(* Logix 5000 project; controller TORQUE Emulate 5570 rev 33.11; software revision 33.00 *)

TASK MainTask (continuous, watchdog 500 ms) : MainProgram, Emulation

MODULES
   Local : Emulate 5570 (ICP 2, rev 33.11)
       : 1756-IB16 (ICP 3, rev 3.1, Input RPI 20 ms)
       : vendor 1 type 7 code 16 (ICP 4, rev 3.1, Output RPI 20 ms)
       : 1756-IF8 (ICP 5, rev 1.1, Input RPI 100 ms)
END_MODULES

PROGRAM Emulation   (* main routine Emulation *)
VAR
   emCROSS_THRD : BOOL;
   emDOWN_SOL_TRAVEL : TIMER := (PRE := 4000);
   emMOTOR1_ONS : BOOL;
   emMOTOR2_ONS : BOOL;
   emMOTOR3_ONS : BOOL;
   emMOTOR4_ONS : BOOL;
   emMOTOR_1_AIN : DINT;
   emMOTOR_1_NO_TORQUE : BOOL;
   emMOTOR_1_OFF_DWELL : TIMER := (PRE := 20);
   emMOTOR_1_ON_DWELL : TIMER := (PRE := 80);
   emMOTOR_2_AIN : DINT;
   emMOTOR_2_ON_DWELL : TIMER := (PRE := 50);
   emMOTOR_3_AIN : DINT;
   emMOTOR_3_ON_DWELL : TIMER := (PRE := 60);
   emMOTOR_4_AIN : DINT;
   emMOTOR_4_CRS_DWELL : TIMER := (PRE := 20);
   emMOTOR_4_ON_DWELL : TIMER := (PRE := 20);
   emNO_TORQUE : BOOL;
   emPART_TRACK : COUNTER := (PRE := 3);
   emSET_POINT : DINT := 97;
END_VAR

ROUTINE Emulation   (* ladder *)
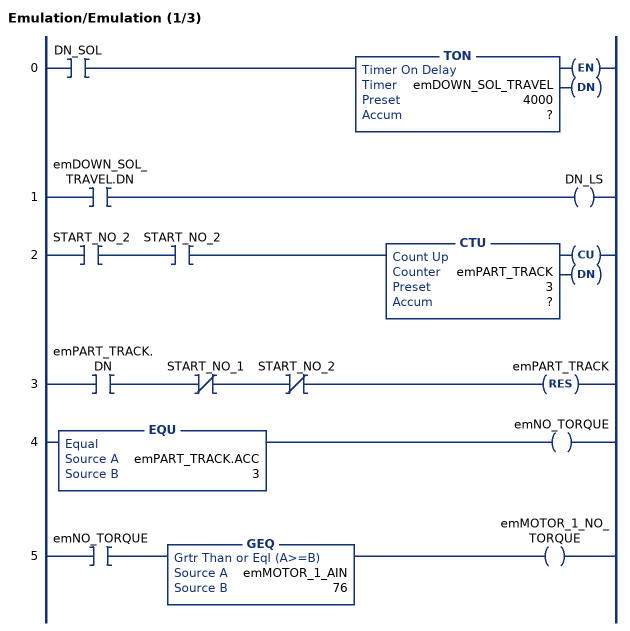
   0: XIC(DN_SOL)TON(emDOWN_SOL_TRAVEL,?,?);
   1: XIC(emDOWN_SOL_TRAVEL.DN)OTE(DN_LS);
   2: XIC(START_NO_2)XIC(START_NO_2)CTU(emPART_TRACK,?,?);
   3: XIC(emPART_TRACK.DN)XIO(START_NO_1)XIO(START_NO_2)RES(emPART_TRACK);
   4: EQU(emPART_TRACK.ACC,3)OTE(emNO_TORQUE);
   5: XIC(emNO_TORQUE)GEQ(emMOTOR_1_AIN,76)OTE(emMOTOR_1_NO_TORQUE);
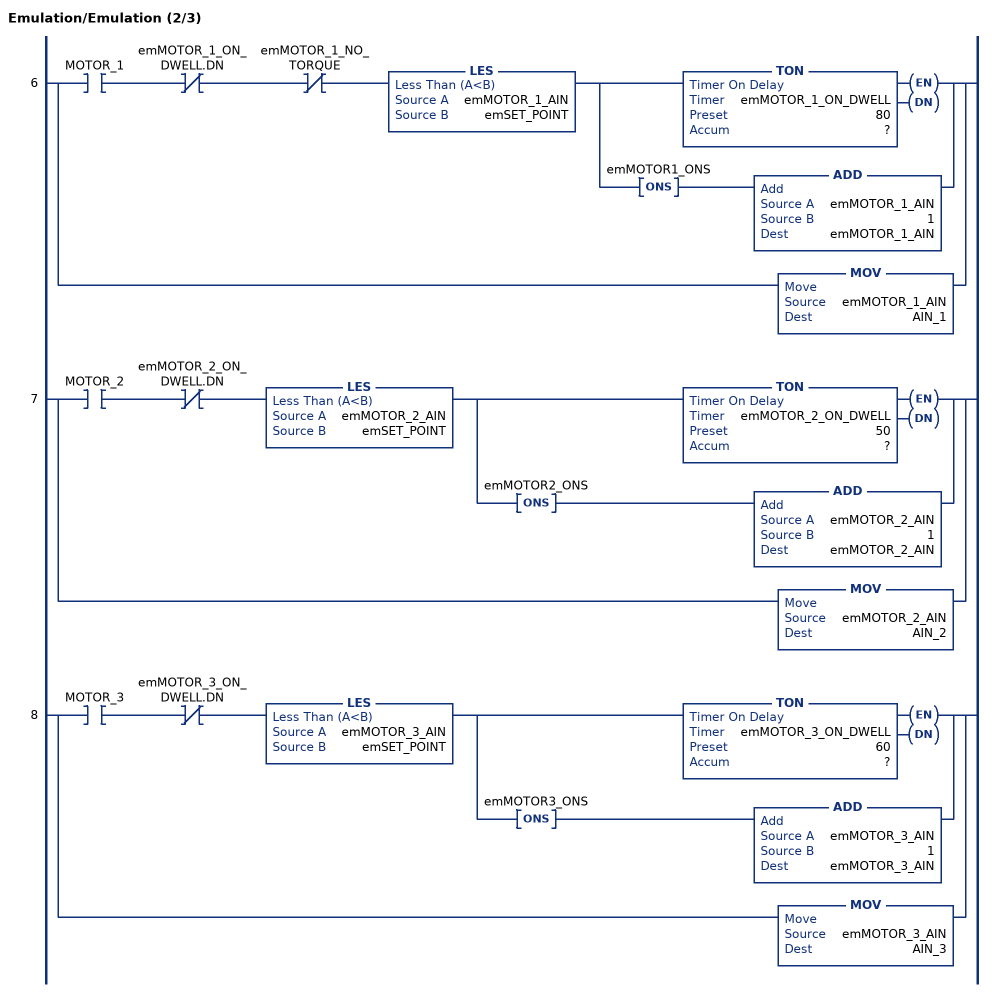
   6: [XIC(MOTOR_1) XIO(emMOTOR_1_ON_DWELL.DN) XIO(emMOTOR_1_NO_TORQUE) LES(emMOTOR_1_AIN,emSET_POINT) [TON(emMOTOR_1_ON_DWELL,?,?) ,ONS(emMOTOR1_ONS) ADD(emMOTOR_1_AIN,1,emMOTOR_1_AIN) ] ,MOV(emMOTOR_1_AIN,AIN_1) ];
   7: [XIC(MOTOR_2) XIO(emMOTOR_2_ON_DWELL.DN) LES(emMOTOR_2_AIN,emSET_POINT) [TON(emMOTOR_2_ON_DWELL,?,?) ,ONS(emMOTOR2_ONS) ADD(emMOTOR_2_AIN,1,emMOTOR_2_AIN) ] ,MOV(emMOTOR_2_AIN,AIN_2) ];
   8: [XIC(MOTOR_3) XIO(emMOTOR_3_ON_DWELL.DN) LES(emMOTOR_3_AIN,emSET_POINT) [TON(emMOTOR_3_ON_DWELL,?,?) ,ONS(emMOTOR3_ONS) ADD(emMOTOR_3_AIN,1,emMOTOR_3_AIN) ] ,MOV(emMOTOR_3_AIN,AIN_3) ];
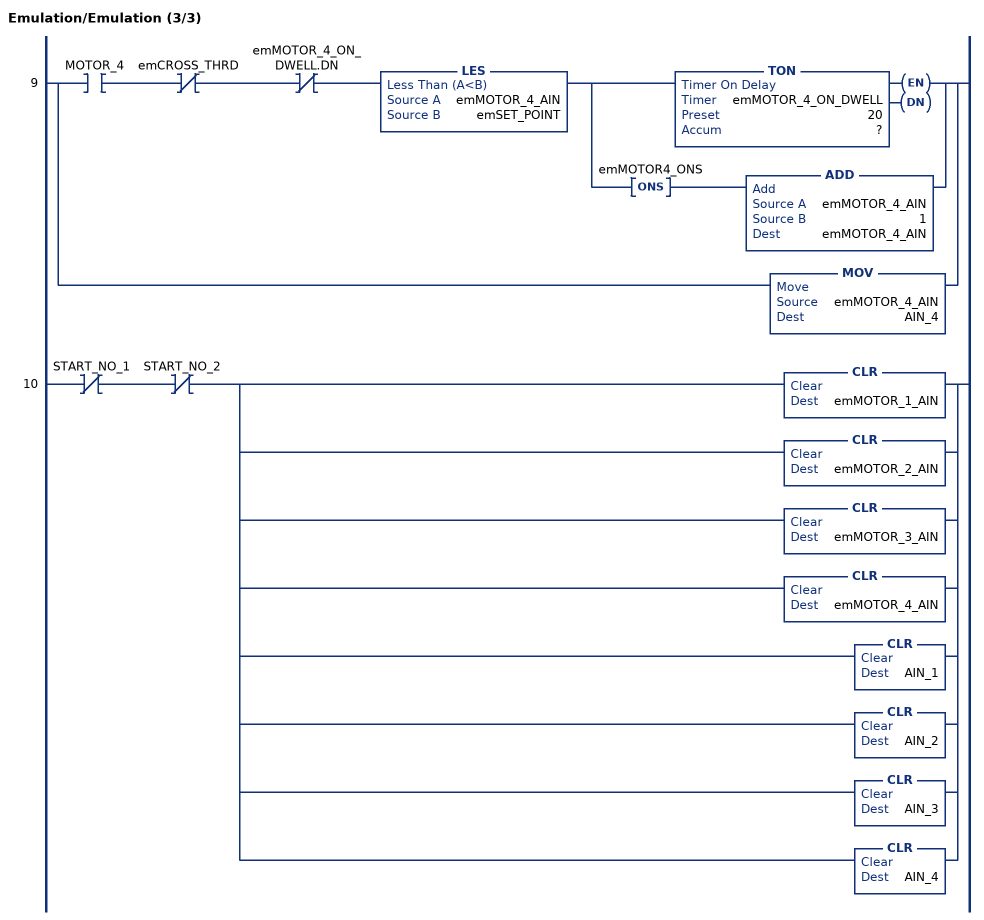
   9: [XIC(MOTOR_4) XIO(emCROSS_THRD) XIO(emMOTOR_4_ON_DWELL.DN) LES(emMOTOR_4_AIN,emSET_POINT) [TON(emMOTOR_4_ON_DWELL,?,?) ,ONS(emMOTOR4_ONS) ADD(emMOTOR_4_AIN,1,emMOTOR_4_AIN) ] ,MOV(emMOTOR_4_AIN,AIN_4) ];
   10: XIO(START_NO_1)XIO(START_NO_2)[CLR(emMOTOR_1_AIN) ,CLR(emMOTOR_2_AIN) ,CLR(emMOTOR_3_AIN) ,CLR(emMOTOR_4_AIN) ,CLR(AIN_1) ,CLR(AIN_2) ,CLR(AIN_3) ,CLR(AIN_4) ];
END_ROUTINE
END_PROGRAM

PROGRAM MainProgram   (* main routine MainRoutine *)

ROUTINE MainRoutine   (* ladder *)
END_ROUTINE
END_PROGRAM
